FUNCTION_BLOCK SUB_LINT (* IEC 61131-3 LINT Subtraction *)
  (* Standard: 61131-3 *)
  (* Version 0.1, 2006-09-11, JHC, Holobloc Inc, Converted to Template. *)
  (* Version 0.0, 2004-12-15, JHC, Rockwell Automation, Converted from SRC format. *)
  (* Compiler header: package fb.rt.plc.math; *)
  (* Compiler classdef: ( IN1 - IN2 ) *)
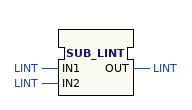
  VAR_INPUT
    IN1 : LINT; (* Minuend *)
    IN2 : LINT; (* Subtrahend *)
  END_VAR
  VAR_OUTPUT
    OUT : LINT; (* Difference *)
  END_VAR
END_FUNCTION_BLOCK
